FUNCTION_BLOCK FB_SituarPale_SFC

VAR_INPUT
    // SFC-Flags
    SFCPause: BOOL;
    SFCReset: BOOL;
    
    // Sincronizacion
    Benido: BOOL ;
    Ejecuta: BOOL;

    // Parametros de tiempo
    //TpoCintaRetenedor: TIME := T#1S;
    
    //TpoPaleSalida: TIME := T#1s;
    //TpoPaleTransferencia: TIME := T#1S;
    
   
    //PulsadorParada AT %I* : BOOL;
    PresenciaPale AT %I* : BOOL;
    
    CodigoPaleBit0 AT %I* : BOOL;
    CodigoPaleBit1 AT  %I* : BOOL;
    CodigoPaleBit2 AT %I* : BOOL;   
    
END_VAR

VAR_OUTPUT
    // Sincronizacion    
    Acabhe: BOOL;
    ListoKalisto: BOOL;
    
    // Parametros de; estado de la estacion
    CodigoPale: BYTE;  
	
	//CintaActiva AT %Q* : BOOL;
   // CintaInvierte AT %Q* : BOOL;
   // RetenedorBaja AT %Q* : BOOL;
    
    //AvisadorSonoro AT %Q* : BOOL;
    
    CintaActiva: BOOL;
    CintaInvierte: BOOL;
    RetenedorBaja: BOOL;
    
    AvisadorSonoro: BOOL;
    
END_VAR
VAR
    TpoPaleEntrada: TIME := T#400MS;
    //CLK: FB_Clock; 
END_VAR

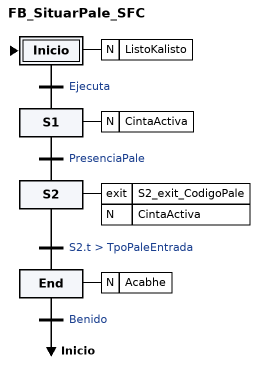
INITIAL_STEP Inicio:
    ListoKalisto(N);
END_STEP
TRANSITION FROM Inicio TO S1
    := Ejecuta;
END_TRANSITION
STEP S1:
    CintaActiva(N);
END_STEP
TRANSITION FROM S1 TO S2
    := PresenciaPale;
END_TRANSITION
STEP S2:
    S2_exit_CodigoPale(P0);  // exit action
    CintaActiva(N);
END_STEP
TRANSITION FROM S2 TO End
    := S2.t > TpoPaleEntrada;
END_TRANSITION
STEP End:
    Acabhe(N);
END_STEP
TRANSITION FROM End TO Inicio
    := Benido;
END_TRANSITION

ACTION S2_exit_CodigoPale:
CodigoPale.0 := CodigoPaleBit0;
CodigoPale.1 := CodigoPaleBit1;
CodigoPale.2 := CodigoPaleBit2;
END_ACTION

END_FUNCTION_BLOCK

(* stored: Version 1.1.0.1, ProductVersion 3.1.4024.12
   POU FB_SituarPale_SFC: Id {161ba697-9c18-4d11-bdbc-4bf04f93ca17}, SpecialFunc None
   Action S2_exit_CodigoPale: Id {f7c3a0d1-d77e-48f7-89c7-36c748650c20} *)
